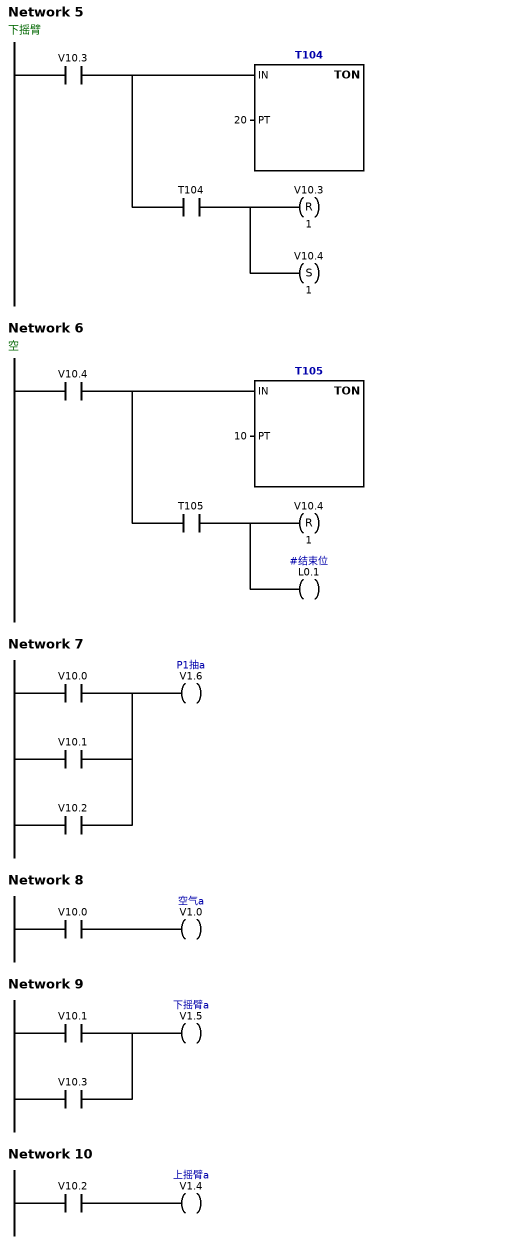
Network 5
// 下摇臂
LD     V10.3
TON    T104, 20
A      T104
R      V10.3, 1
S      V10.4, 1
Network 6
// 空
LD     V10.4
TON    T105, 10
A      T105
R      V10.4, 1
=      #结束位:L0.1
Network 7
LD     V10.0
O      V10.1
O      V10.2
=      P1抽a:V1.6
Network 8
LD     V10.0
=      空气a:V1.0
Network 9
LD     V10.1
O      V10.3
=      下摇臂a:V1.5
Network 10
LD     V10.2
=      上摇臂a:V1.4
END_SUBROUTINE_BLOCK

SUBROUTINE_BLOCK M排空:SBR5
TITLE=P1抽取比色皿内液体
VAR_INPUT
时间:WORD;	// LW0 
END_VAR
VAR_IN_OUT
启动位:BOOL;	// L2.0 
END_VAR
VAR_OUTPUT
结束位:BOOL;	// L2.1 
END_VAR
BEGIN
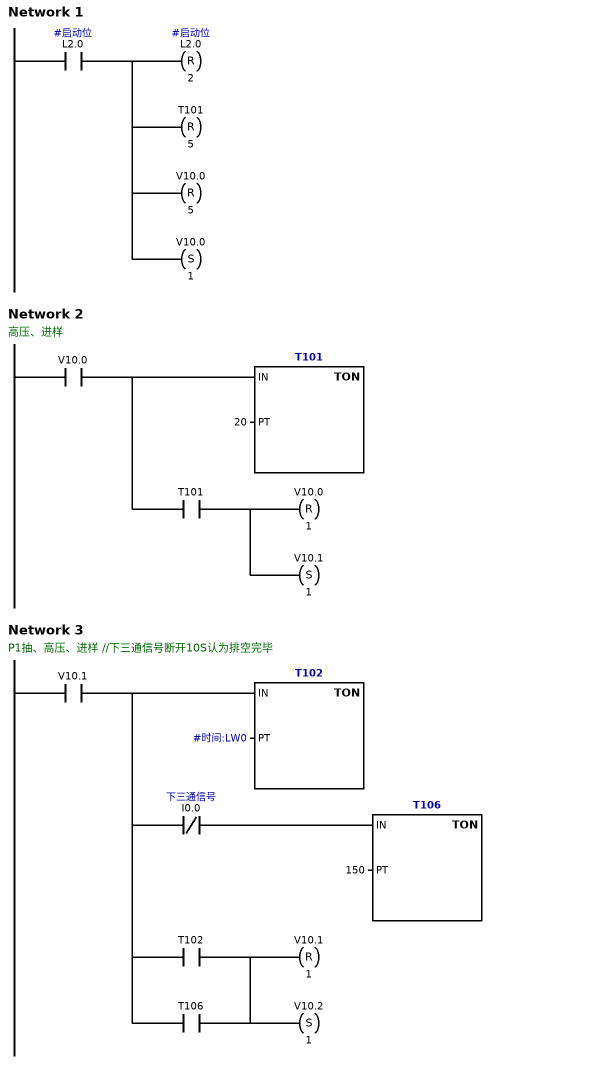
Network 1
LD     #启动位:L2.0
R      #启动位:L2.0, 2
R      T101, 5
R      V10.0, 5
S      V10.0, 1
Network 2
// 高压、进样
LD     V10.0
TON    T101, 20
A      T101
R      V10.0, 1
S      V10.1, 1
Network 3
// P1抽、高压、进样 //下三通信号断开10S认为排空完毕
LD     V10.1
LPS
TON    T102, #时间:LW0
AN     下三通信号:I0.0
TON    T106, 150
LPP
LD     T102
O      T106
ALD
R      V10.1, 1
S      V10.2, 1
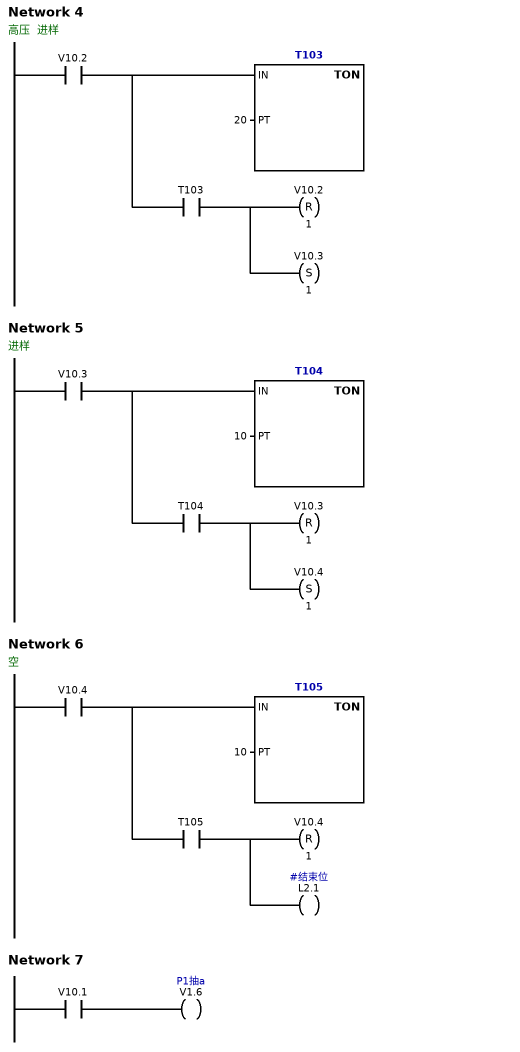
Network 4
// 高压  进样  
LD     V10.2
TON    T103, 20
A      T103
R      V10.2, 1
S      V10.3, 1
Network 5
// 进样  
LD     V10.3
TON    T104, 10
A      T104
R      V10.3, 1
S      V10.4, 1
Network 6
// 空
LD     V10.4
TON    T105, 10
A      T105
R      V10.4, 1
=      #结束位:L2.1
Network 7
LD     V10.1
=      P1抽a:V1.6
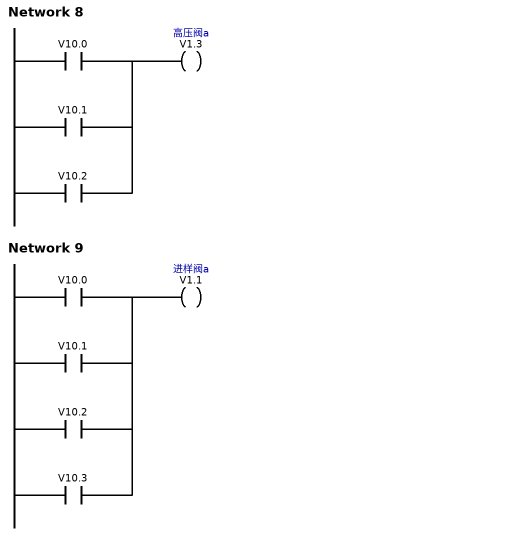
Network 8
LD     V10.0
O      V10.1
O      V10.2
=      高压阀a:V1.3
Network 9
LD     V10.0
O      V10.1
O      V10.2
O      V10.3
=      进样阀a:V1.1
END_SUBROUTINE_BLOCK

SUBROUTINE_BLOCK M润洗:SBR6
TITLE=
VAR_INPUT
抽液时间:WORD;	// LW0 
抽空时间:WORD;	// LW2 
END_VAR
VAR_IN_OUT
启动位:BOOL;	// L4.0 
END_VAR
VAR_OUTPUT
结束位:BOOL;	// L4.1 
采样阀:BOOL;	// L4.2 
END_VAR
BEGIN
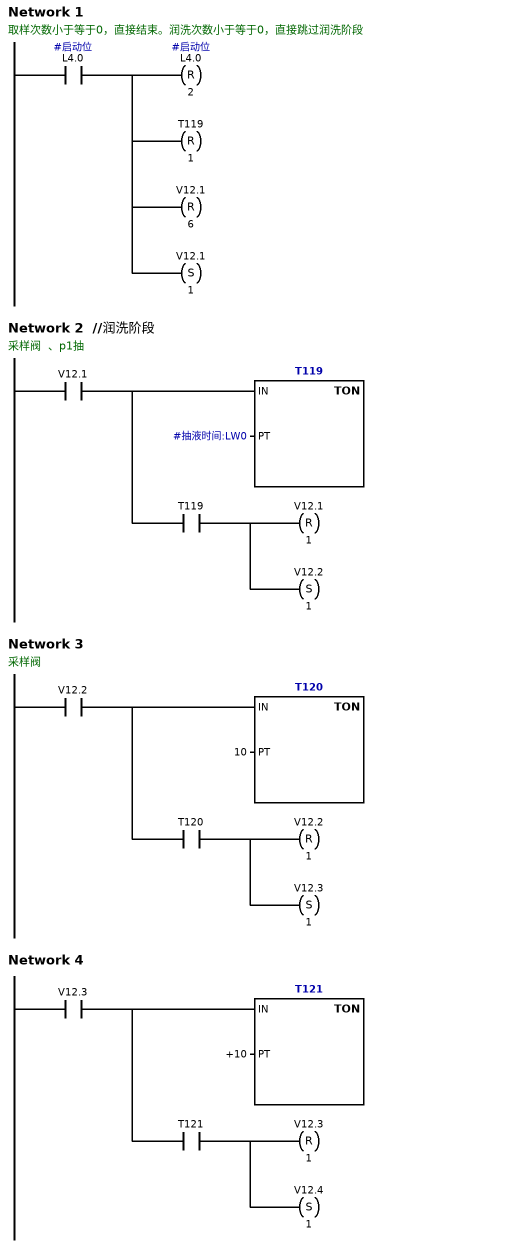
Network 1
// 取样次数小于等于0，直接结束。润洗次数小于等于0，直接跳过润洗阶段
LD     #启动位:L4.0
R      #启动位:L4.0, 2
R      T119, 1
R      V12.1, 6
S      V12.1, 1
Network 2 // //润洗阶段
// 采样阀  、p1抽
LD     V12.1
TON    T119, #抽液时间:LW0
A      T119
R      V12.1, 1
S      V12.2, 1
Network 3
//  采样阀
LD     V12.2
TON    T120, 10
A      T120
R      V12.2, 1
S      V12.3, 1
Network 4
LD     V12.3
TON    T121, +10
A      T121
R      V12.3, 1
S      V12.4, 1
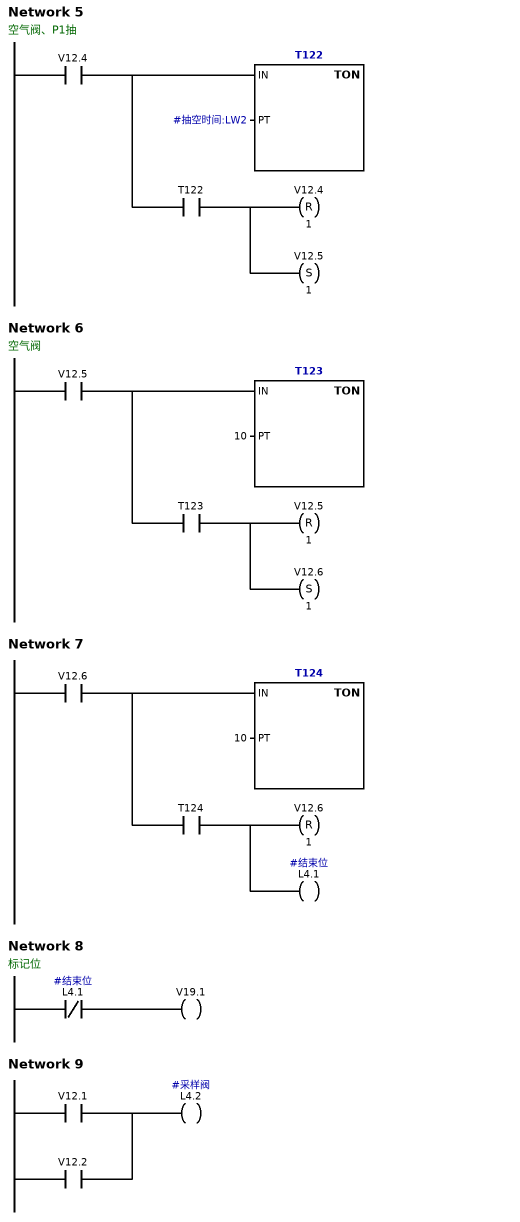
Network 5
// 空气阀、P1抽
LD     V12.4
TON    T122, #抽空时间:LW2
A      T122
R      V12.4, 1
S      V12.5, 1
Network 6
// 空气阀
LD     V12.5
TON    T123, 10
A      T123
R      V12.5, 1
S      V12.6, 1
Network 7
LD     V12.6
TON    T124, 10
A      T124
R      V12.6, 1
=      #结束位:L4.1
Network 8
// 标记位
LDN    #结束位:L4.1
=      V19.1
Network 9
LD     V12.1
O      V12.2
=      #采样阀:L4.2
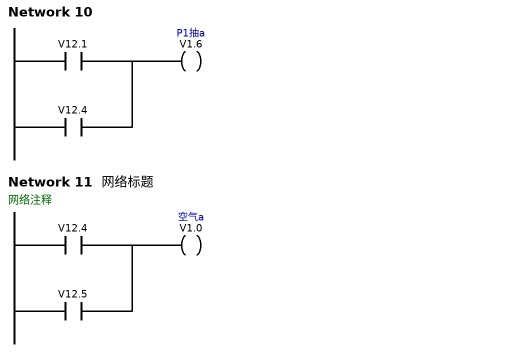
Network 10
LD     V12.1
O      V12.4
=      P1抽a:V1.6
Network 11 // 网络标题
// 网络注释
LD     V12.4
O      V12.5
=      空气a:V1.0
Network 13 // 网络标题
// 网络注释
END_SUBROUTINE_BLOCK

SUBROUTINE_BLOCK 【流程】:SBR7
TITLE=
VAR_IN_OUT
启动位:BOOL;	// L0.0 
END_VAR
VAR_OUTPUT
结束位:BOOL;	// L0.1 
END_VAR
BEGIN
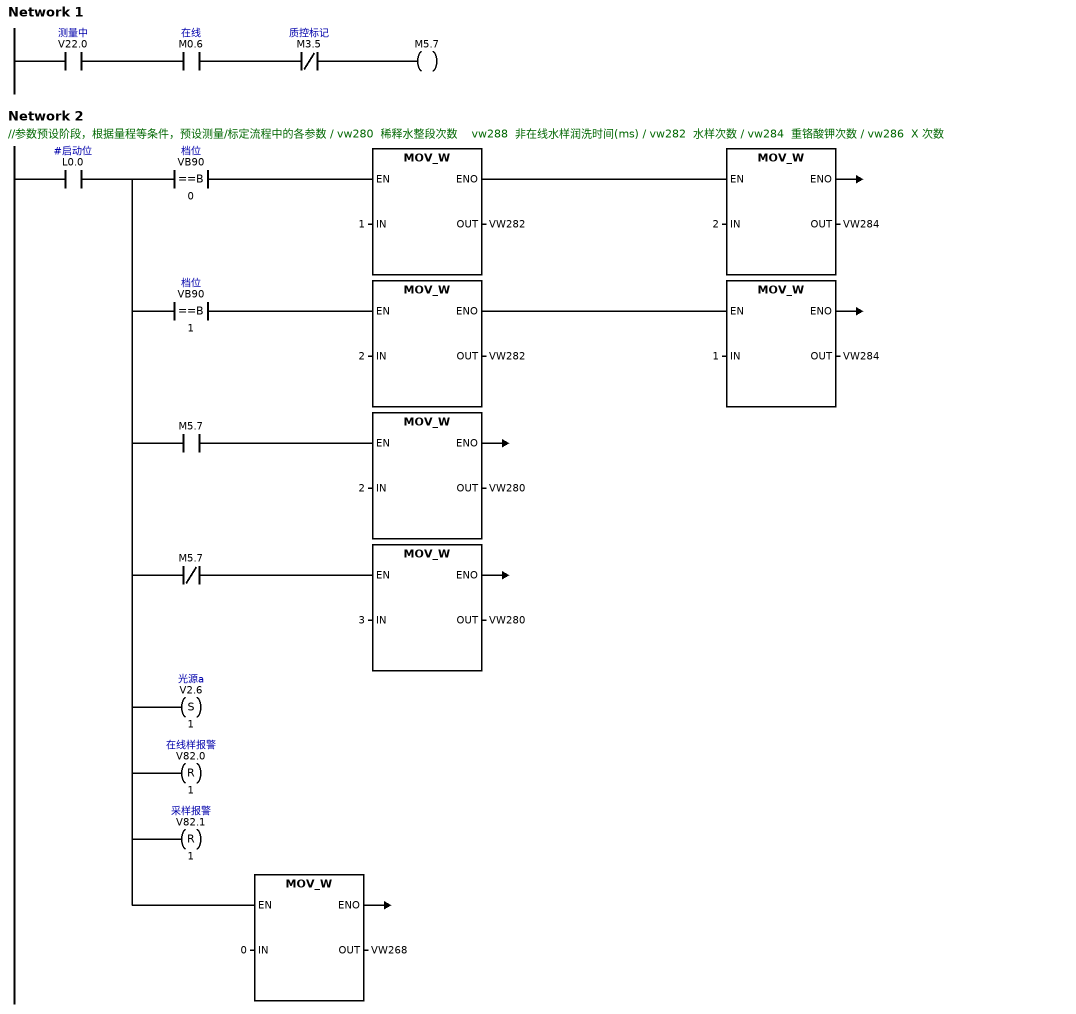
Network 1
LD     测量中:V22.0
A      在线:M0.6
AN     质控标记:M3.5
=      M5.7
Network 2
// //参数预设阶段，根据量程等条件，预设测量/标定流程中的各参数
// vw280  稀释水整段次数    vw288  非在线水样润洗时间(ms)
// vw282  水样次数
// vw284  重铬酸钾次数
// vw286  X 次数
LD     #启动位:L0.0
LPS
AB=    档位:VB90, 0
MOVW   1, VW282
AENO
MOVW   2, VW284
LRD
AB=    档位:VB90, 1
MOVW   2, VW282
AENO
MOVW   1, VW284
LRD
A      M5.7
MOVW   2, VW280
LRD
AN     M5.7
MOVW   3, VW280
LRD
S      光源a:V2.6, 1
LRD
R      在线样报警:V82.0, 1
LRD
R      采样报警:V82.1, 1
LPP
MOVW   0, VW268
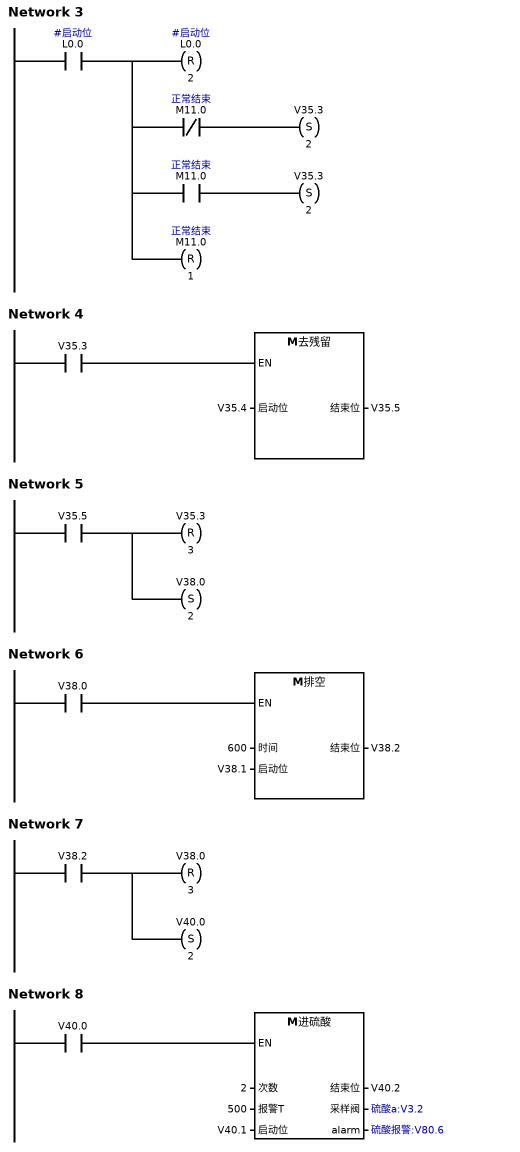
Network 3
LD     #启动位:L0.0
LPS
R      #启动位:L0.0, 2
AN     正常结束:M11.0
S      V35.3, 2
LRD
A      正常结束:M11.0
S      V35.3, 2
LPP
R      正常结束:M11.0, 1
Network 4
LD     V35.3
CALL   M去残留:SBR4, V35.4, V35.5
Network 5
LD     V35.5
R      V35.3, 3
S      V38.0, 2
Network 6
LD     V38.0
CALL   M排空:SBR5, 600, V38.1, V38.2
Network 7
LD     V38.2
R      V38.0, 3
S      V40.0, 2
Network 8
LD     V40.0
CALL   M进硫酸:SBR3, 2, 500, V40.1, V40.2, 硫酸a:V3.2, 硫酸报警:V80.6
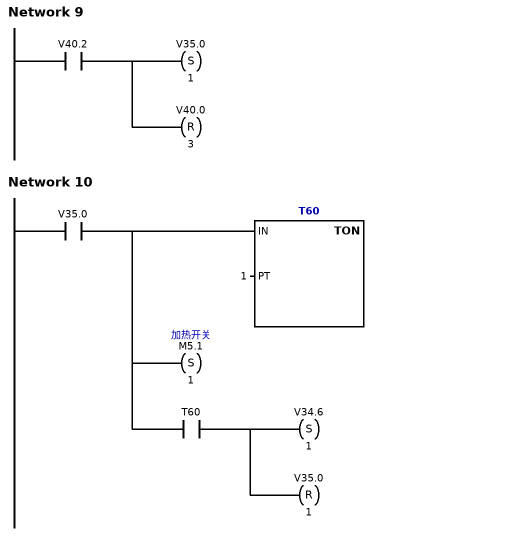
Network 9
LD     V40.2
S      V35.0, 1
R      V40.0, 3
Network 10
LD     V35.0
TON    T60, 1
S      加热开关:M5.1, 1
A      T60
S      V34.6, 1
R      V35.0, 1
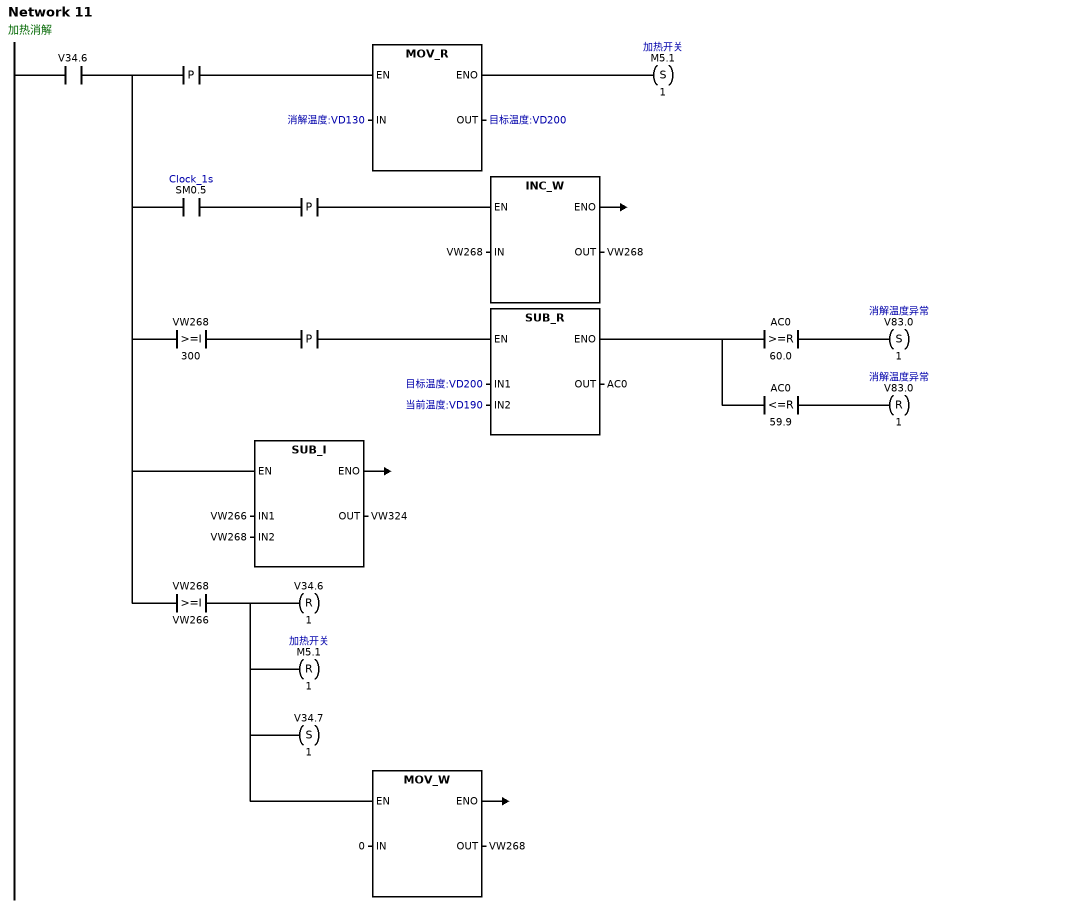
Network 11
// 加热消解
LD     V34.6
LPS
EU
MOVR   消解温度:VD130, 目标温度:VD200
AENO
S      加热开关:M5.1, 1
LRD
A      Clock_1s:SM0.5
EU
INCW   VW268
LRD
AW>=   VW268, 300
EU
MOVR   目标温度:VD200, AC0
AENO
-R     当前温度:VD190, AC0
AENO
LPS
AR>=   AC0, 60.0
S      消解温度异常:V83.0, 1
LPP
AR<=   AC0, 59.9
R      消解温度异常:V83.0, 1
LRD
MOVW   VW266, VW324
-I     VW268, VW324
LPP
AW>=   VW268, VW266
R      V34.6, 1
R      加热开关:M5.1, 1
S      V34.7, 1
MOVW   0, VW268
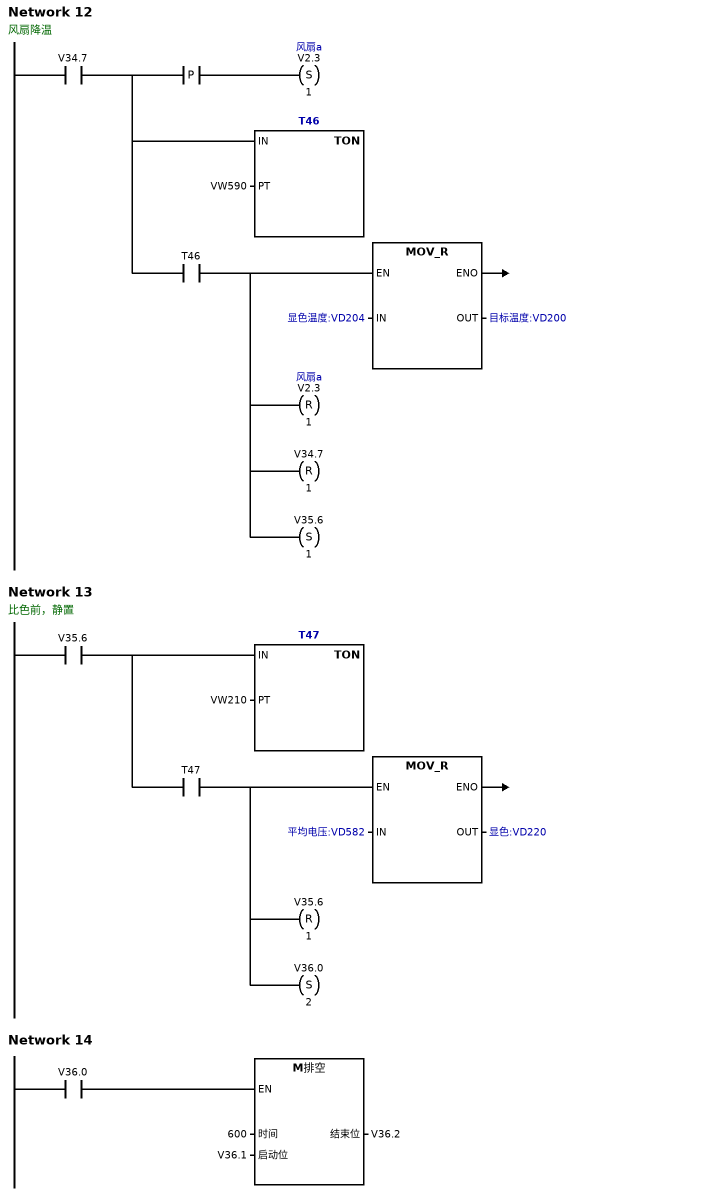
Network 12
// 风扇降温   
// (network saved uncompiled; LAD cells follow)
// row 0: c0 -| |- V34.7 v  c1 -|P|-  c2 -(S) 风扇a:V2.3, 1
// row 1: c0 ^v  c1 --  c2 [TON T46 IN:=power@row1, PT:=VW590]
// row 2: c0 ^v  c2 [box]
// row 3: c0 ^  c1 -| |- T46 v  c2 --  c3 [MOV_R EN:=power@row3, IN:=显色温度:VD204, ENO=>power, OUT=>目标温度:VD200]  c4 ->
// row 4: c1 ^v  c3 [box]
// row 5: c1 ^v  c2 -(R) 风扇a:V2.3, 1
// row 6: c1 ^v  c2 -(R) V34.7, 1
// row 7: c1 ^  c2 -(S) V35.6, 1
Network 13
// 比色前，静置
LD     V35.6
TON    T47, VW210
A      T47
MOVR   平均电压:VD582, 显色:VD220
R      V35.6, 1
S      V36.0, 2
Network 14
LD     V36.0
CALL   M排空:SBR5, 600, V36.1, V36.2
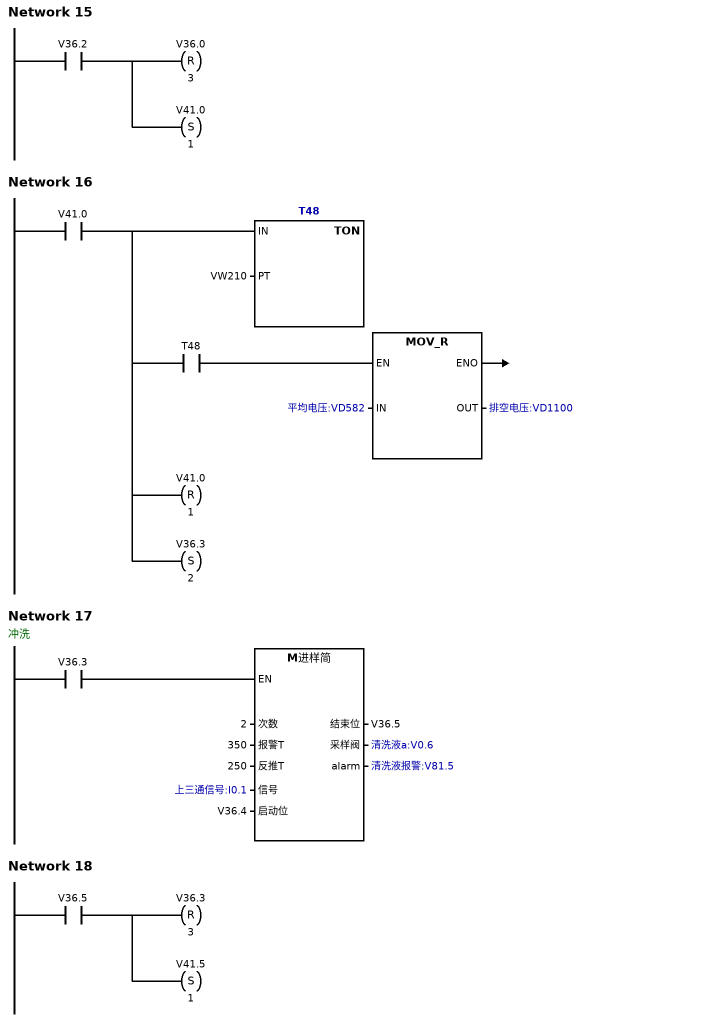
Network 15
LD     V36.2
R      V36.0, 3
S      V41.0, 1
Network 16
LD     V41.0
LPS
TON    T48, VW210
A      T48
MOVR   平均电压:VD582, 排空电压:VD1100
LRD
R      V41.0, 1
LPP
S      V36.3, 2
Network 17
// 冲洗
LD     V36.3
CALL   M进样简:SBR1, 2, 350, 250, 上三通信号:I0.1, V36.4, V36.5, 清洗液a:V0.6, 清洗液报警:V81.5
Network 18
LD     V36.5
R      V36.3, 3
S      V41.5, 1
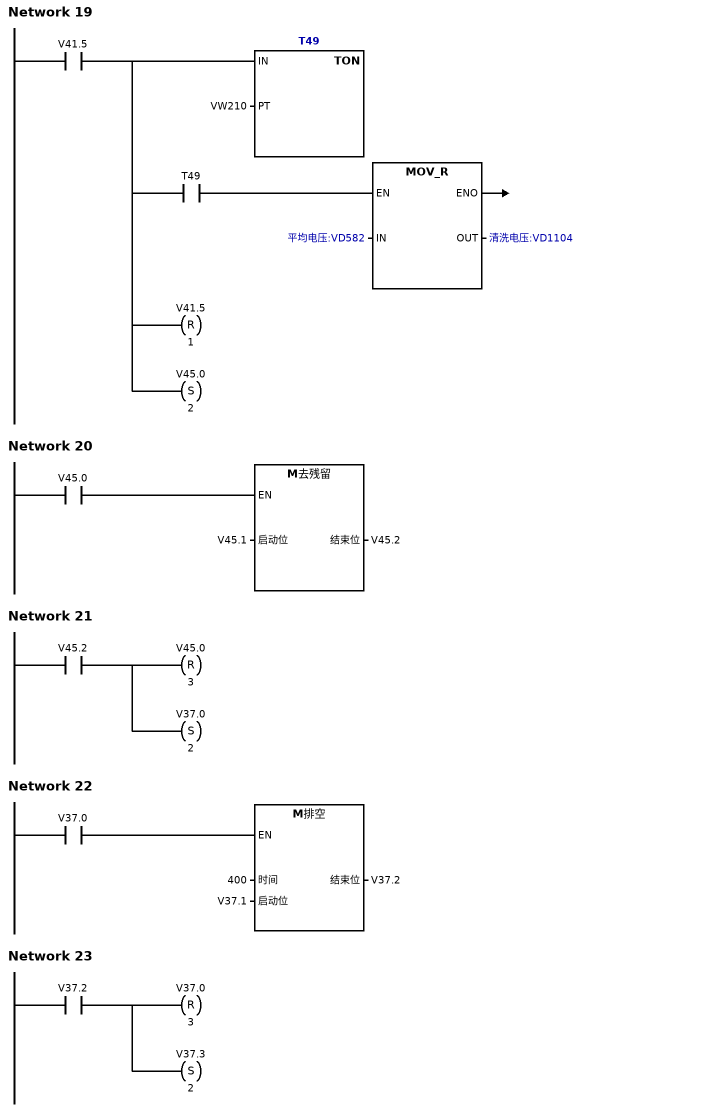
Network 19
LD     V41.5
LPS
TON    T49, VW210
A      T49
MOVR   平均电压:VD582, 清洗电压:VD1104
LRD
R      V41.5, 1
LPP
S      V45.0, 2
Network 20
LD     V45.0
CALL   M去残留:SBR4, V45.1, V45.2
Network 21
LD     V45.2
R      V45.0, 3
S      V37.0, 2
Network 22
LD     V37.0
CALL   M排空:SBR5, 400, V37.1, V37.2
Network 23
LD     V37.2
R      V37.0, 3
S      V37.3, 2
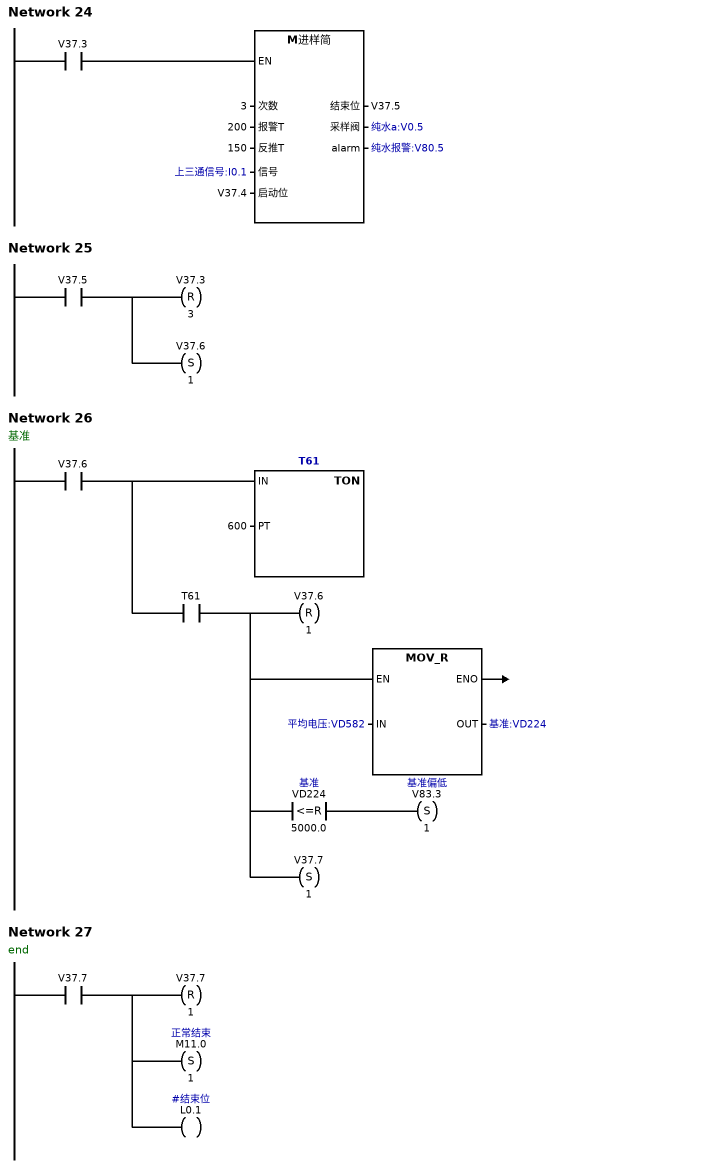
Network 24
LD     V37.3
CALL   M进样简:SBR1, 3, 200, 150, 上三通信号:I0.1, V37.4, V37.5, 纯水a:V0.5, 纯水报警:V80.5
Network 25
LD     V37.5
R      V37.3, 3
S      V37.6, 1
Network 26
// 基准
LD     V37.6
TON    T61, 600
A      T61
LPS
R      V37.6, 1
MOVR   平均电压:VD582, 基准:VD224
AR<=   基准:VD224, 5000.0
S      基准偏低:V83.3, 1
LPP
S      V37.7, 1
Network 27
// end
LD     V37.7
R      V37.7, 1
S      正常结束:M11.0, 1
=      #结束位:L0.1
END_SUBROUTINE_BLOCK

SUBROUTINE_BLOCK 输出Q:SBR8
TITLE=
BEGIN
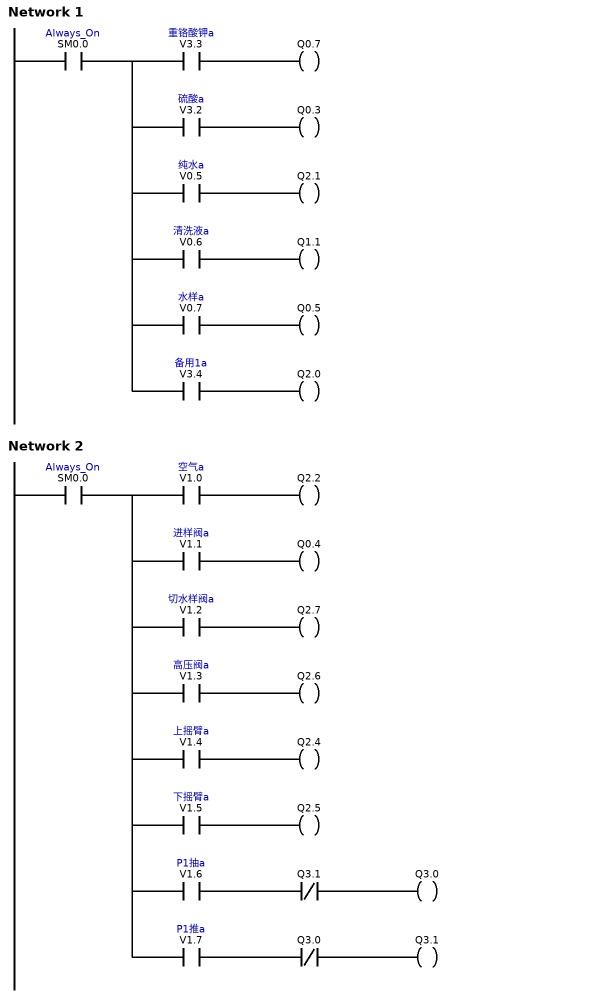
Network 1
LD     Always_On:SM0.0
LPS
A      重铬酸钾a:V3.3
=      Q0.7
LRD
A      硫酸a:V3.2
=      Q0.3
LRD
A      纯水a:V0.5
=      Q2.1
LRD
A      清洗液a:V0.6
=      Q1.1
LRD
A      水样a:V0.7
=      Q0.5
LPP
A      备用1a:V3.4
=      Q2.0
Network 2
LD     Always_On:SM0.0
LPS
A      空气a:V1.0
=      Q2.2
LRD
A      进样阀a:V1.1
=      Q0.4
LRD
A      切水样阀a:V1.2
=      Q2.7
LRD
A      高压阀a:V1.3
=      Q2.6
LRD
A      上摇臂a:V1.4
=      Q2.4
LRD
A      下摇臂a:V1.5
=      Q2.5
LRD
A      P1抽a:V1.6
AN     Q3.1
=      Q3.0
LPP
A      P1推a:V1.7
AN     Q3.0
=      Q3.1
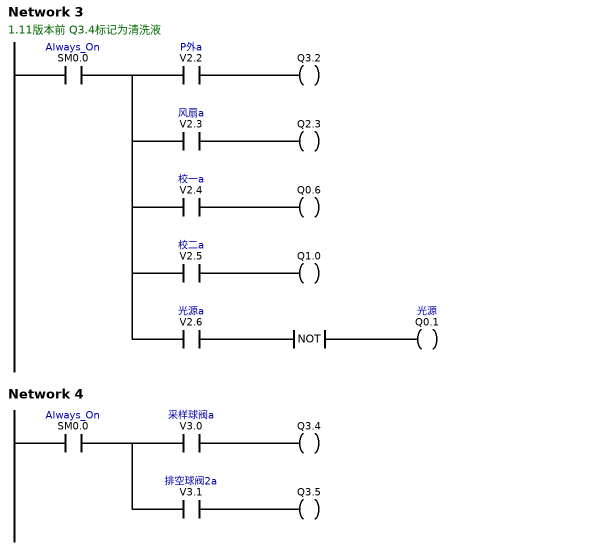
Network 3
// 1.11版本前 Q3.4标记为清洗液  
LD     Always_On:SM0.0
LPS
A      P外a:V2.2
=      Q3.2
LRD
A      风扇a:V2.3
=      Q2.3
LRD
A      校一a:V2.4
=      Q0.6
LRD
A      校二a:V2.5
=      Q1.0
LPP
A      光源a:V2.6
NOT
=      光源:Q0.1
Network 4
LD     Always_On:SM0.0
LPS
A      采样球阀a:V3.0
=      Q3.4
LPP
A      排空球阀2a:V3.1
=      Q3.5
END_SUBROUTINE_BLOCK

SUBROUTINE_BLOCK PID计算:SBR9
TITLE=子程序注释
VAR_INPUT
当前温度:REAL;	// LD0 
目标温度:REAL;	// LD4 
END_VAR
VAR_OUTPUT
占空比:INT;	// LW8 
END_VAR
VAR
温度差:REAL;	// LD10 
END_VAR
BEGIN
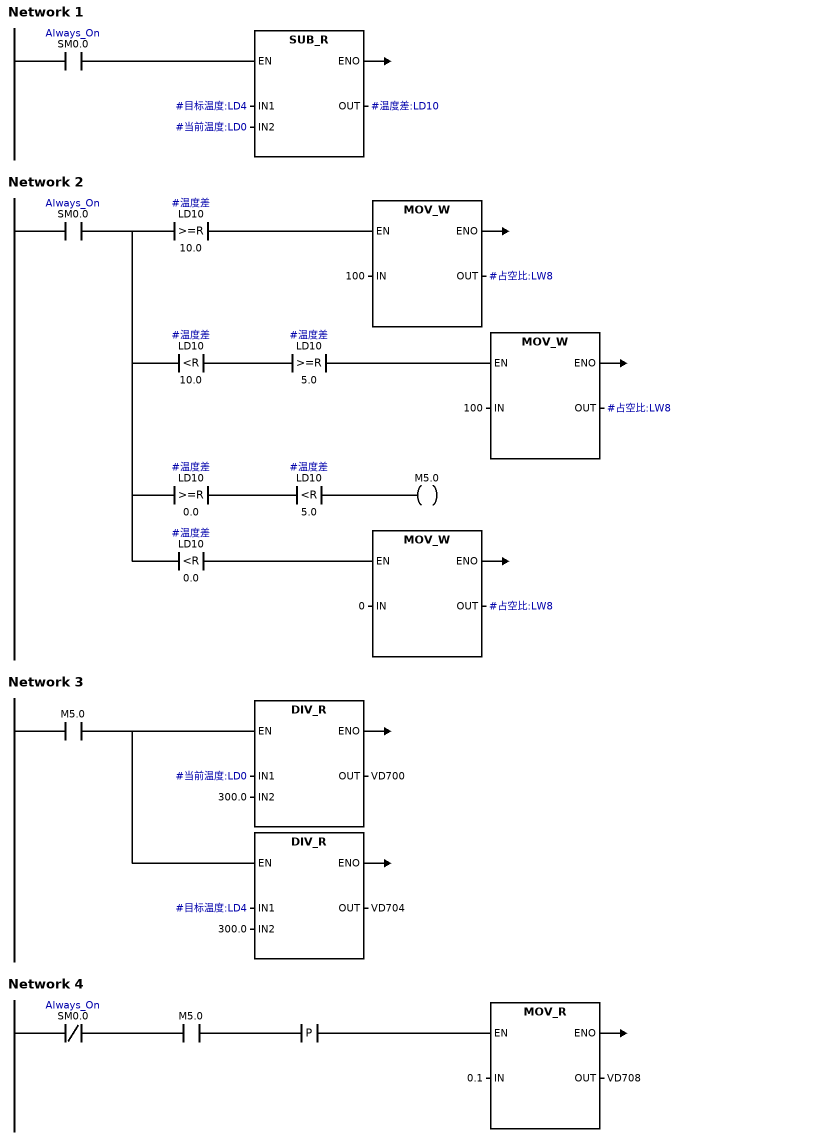
Network 1
LD     Always_On:SM0.0
MOVR   #目标温度:LD4, #温度差:LD10
-R     #当前温度:LD0, #温度差:LD10
Network 2
LD     Always_On:SM0.0
LPS
AR>=   #温度差:LD10, 10.0
MOVW   100, #占空比:LW8
LRD
AR<    #温度差:LD10, 10.0
AR>=   #温度差:LD10, 5.0
MOVW   100, #占空比:LW8
LRD
AR>=   #温度差:LD10, 0.0
AR<    #温度差:LD10, 5.0
=      M5.0
LPP
AR<    #温度差:LD10, 0.0
MOVW   0, #占空比:LW8
Network 3
LD     M5.0
MOVR   #当前温度:LD0, VD700
/R     300.0, VD700
MOVR   #目标温度:LD4, VD704
/R     300.0, VD704
Network 4
LDN    Always_On:SM0.0
A      M5.0
EU
MOVR   0.1, VD708
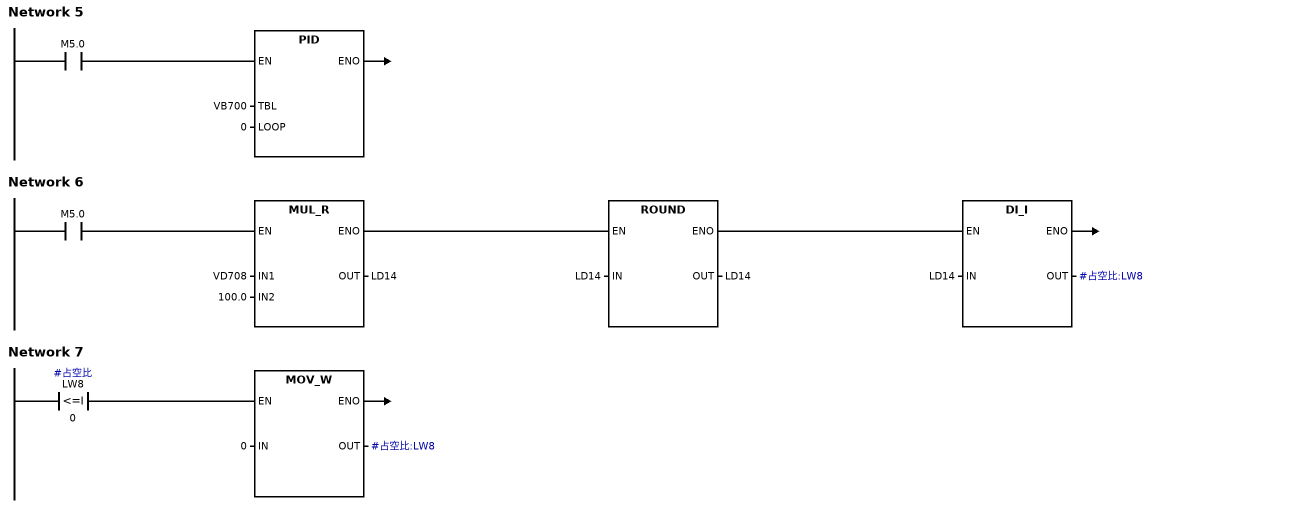
Network 5
LD     M5.0
PID    VB700, 0
Network 6
LD     M5.0
MOVR   VD708, LD14
AENO
*R     100.0, LD14
AENO
ROUND  LD14, LD14
AENO
DTI    LD14, #占空比:LW8
Network 7
LDW<=  #占空比:LW8, 0
MOVW   0, #占空比:LW8
END_SUBROUTINE_BLOCK

SUBROUTINE_BLOCK 二层:SBR10
TITLE=子程序注释
BEGIN
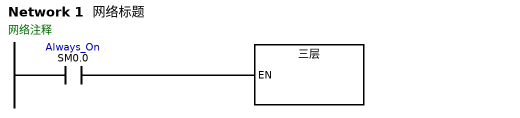
Network 1 // 网络标题
// 网络注释
LD     Always_On:SM0.0
CALL   三层:SBR36
END_SUBROUTINE_BLOCK

SUBROUTINE_BLOCK KBA:SBR11
TITLE=子程序注释
VAR_INPUT
显色1:REAL;	// LD0 
基准1:REAL;	// LD4 
浓度1:REAL;	// LD8 
显色2:REAL;	// LD12 
基准2:REAL;	// LD16 
浓度2:REAL;	// LD20 
END_VAR
VAR_OUTPUT
A1:REAL;	// LD24 
A2:REAL;	// LD28 
K:REAL;	// LD32 
b:REAL;	// LD36 
END_VAR
BEGIN
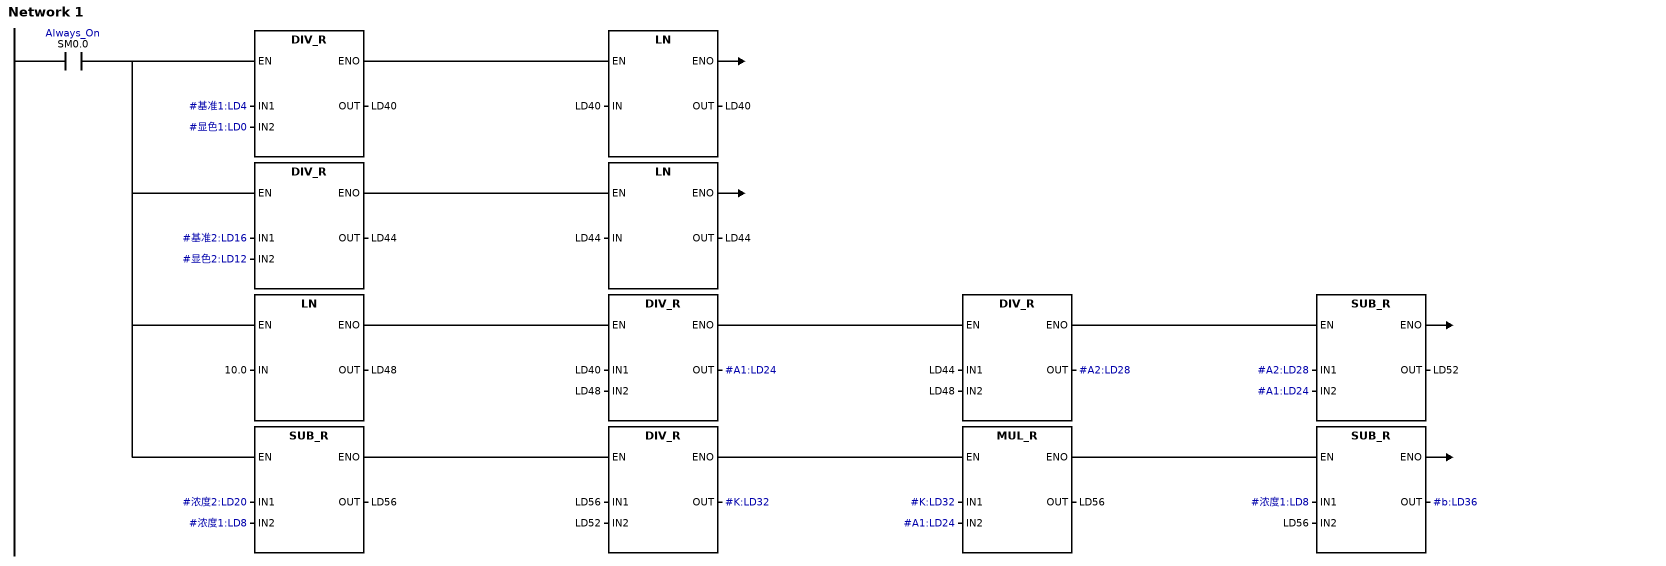
Network 1
LD     Always_On:SM0.0
LPS
MOVR   #基准1:LD4, LD40
AENO
/R     #显色1:LD0, LD40
AENO
LN     LD40, LD40
LRD
MOVR   #基准2:LD16, LD44
AENO
/R     #显色2:LD12, LD44
AENO
LN     LD44, LD44
LRD
LN     10.0, LD48
AENO
MOVR   LD40, #A1:LD24
AENO
/R     LD48, #A1:LD24
AENO
MOVR   LD44, #A2:LD28
AENO
/R     LD48, #A2:LD28
AENO
MOVR   #A2:LD28, LD52
-R     #A1:LD24, LD52
LPP
MOVR   #浓度2:LD20, LD56
AENO
-R     #浓度1:LD8, LD56
AENO
MOVR   LD56, #K:LD32
AENO
/R     LD52, #K:LD32
AENO
MOVR   #K:LD32, LD56
AENO
*R     #A1:LD24, LD56
AENO
MOVR   #浓度1:LD8, #b:LD36
-R     LD56, #b:LD36
Network 2 // 网络标题
// 网络注释
END_SUBROUTINE_BLOCK

SUBROUTINE_BLOCK 间隔测量:SBR12
TITLE=子程序注释
BEGIN
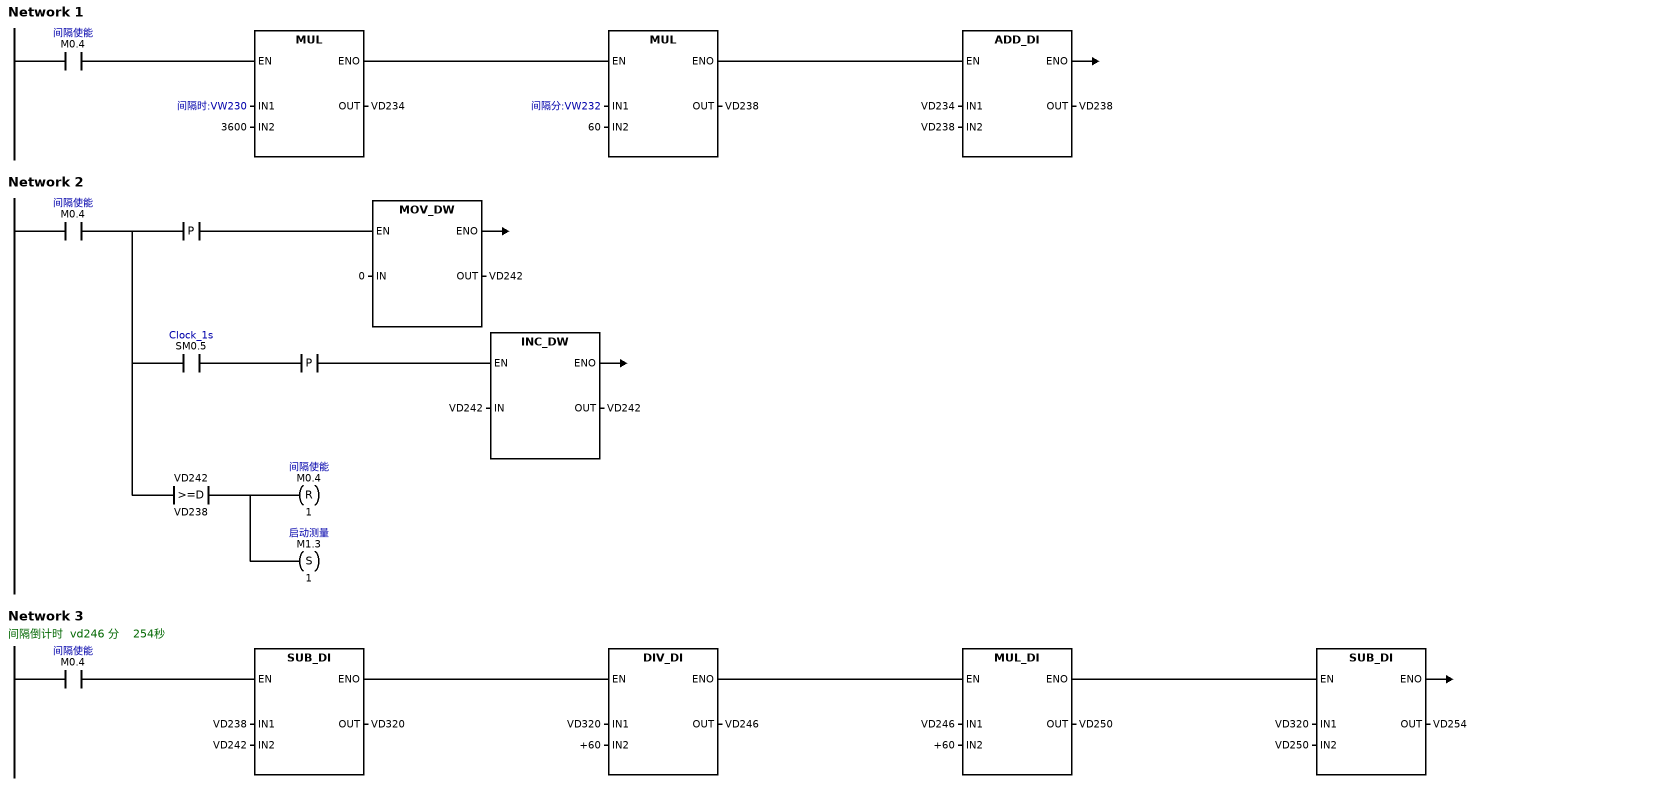
Network 1
LD     间隔使能:M0.4
MOVW   间隔时:VW230, VW236
AENO
MUL    3600, VD234
AENO
MOVW   间隔分:VW232, VW240
AENO
MUL    60, VD238
AENO
+D     VD234, VD238
Network 2
LD     间隔使能:M0.4
LPS
EU
MOVD   0, VD242
LRD
A      Clock_1s:SM0.5
EU
INCD   VD242
LPP
AD>=   VD242, VD238
R      间隔使能:M0.4, 1
S      启动测量:M1.3, 1
Network 3
// 间隔倒计时  vd246 分    254秒
LD     间隔使能:M0.4
MOVD   VD238, VD320
AENO
-D     VD242, VD320
AENO
MOVD   VD320, VD246
AENO
/D     +60, VD246
AENO
MOVD   VD246, VD250
AENO
*D     +60, VD250
AENO
MOVD   VD320, VD254
-D     VD250, VD254
Network 4 // 网络标题
// 网络注释
END_SUBROUTINE_BLOCK

SUBROUTINE_BLOCK 整点测量:SBR13
TITLE=子程序注释
BEGIN
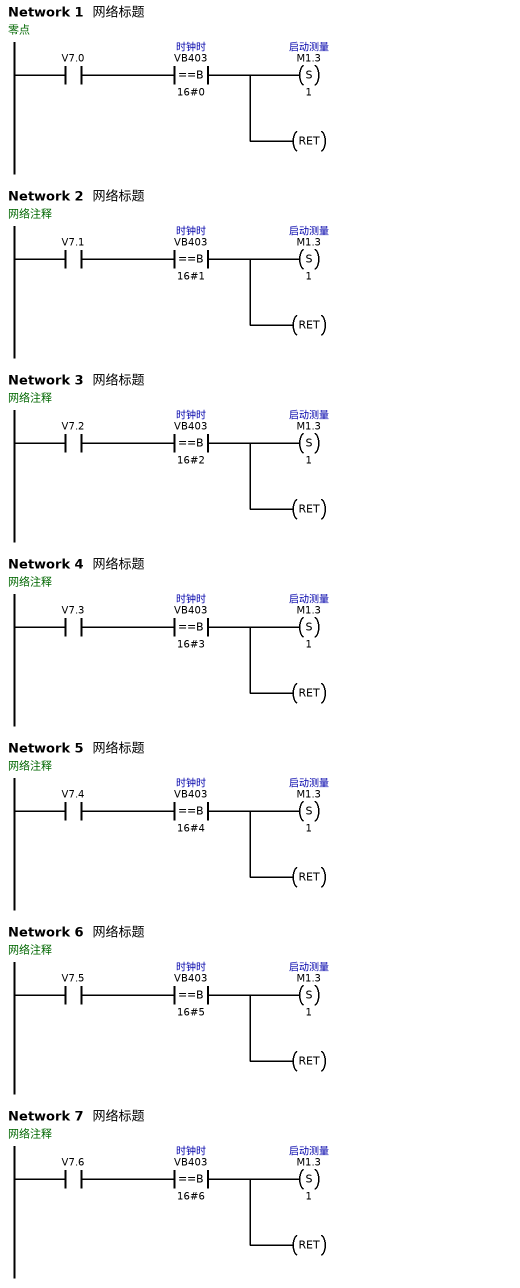
Network 1 // 网络标题
// 零点
LD     V7.0
AB=    时钟时:VB403, 16#0
S      启动测量:M1.3, 1
CRET
Network 2 // 网络标题
// 网络注释
LD     V7.1
AB=    时钟时:VB403, 16#1
S      启动测量:M1.3, 1
CRET
Network 3 // 网络标题
// 网络注释
LD     V7.2
AB=    时钟时:VB403, 16#2
S      启动测量:M1.3, 1
CRET
Network 4 // 网络标题
// 网络注释
LD     V7.3
AB=    时钟时:VB403, 16#3
S      启动测量:M1.3, 1
CRET
Network 5 // 网络标题
// 网络注释
LD     V7.4
AB=    时钟时:VB403, 16#4
S      启动测量:M1.3, 1
CRET
Network 6 // 网络标题
// 网络注释
LD     V7.5
AB=    时钟时:VB403, 16#5
S      启动测量:M1.3, 1
CRET
Network 7 // 网络标题
// 网络注释
LD     V7.6
AB=    时钟时:VB403, 16#6
S      启动测量:M1.3, 1
CRET
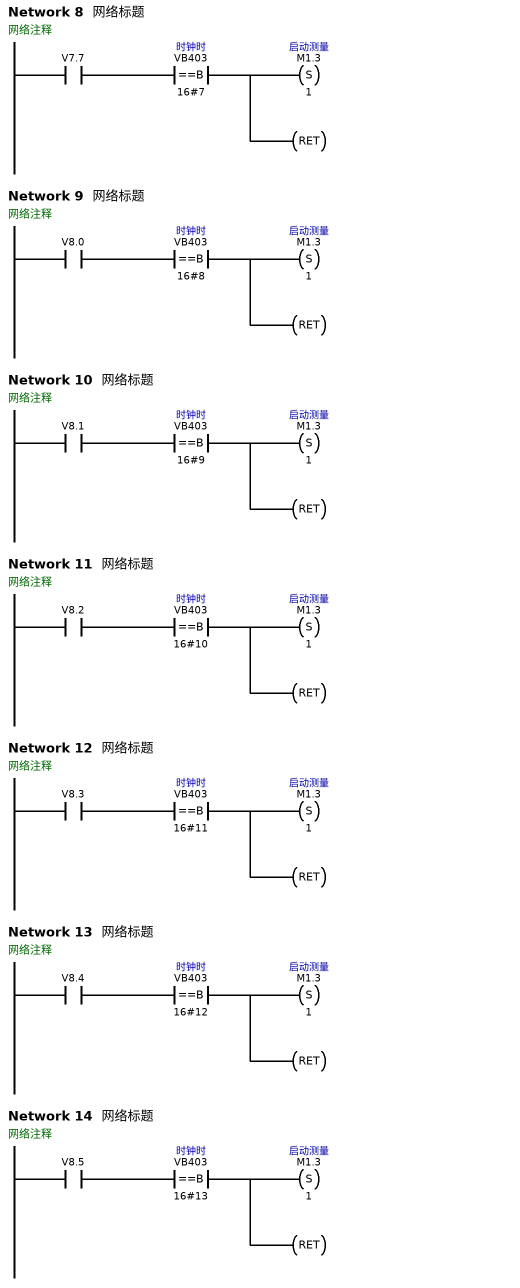
Network 8 // 网络标题
// 网络注释
LD     V7.7
AB=    时钟时:VB403, 16#7
S      启动测量:M1.3, 1
CRET
Network 9 // 网络标题
// 网络注释
LD     V8.0
AB=    时钟时:VB403, 16#8
S      启动测量:M1.3, 1
CRET
Network 10 // 网络标题
// 网络注释
LD     V8.1
AB=    时钟时:VB403, 16#9
S      启动测量:M1.3, 1
CRET
Network 11 // 网络标题
// 网络注释
LD     V8.2
AB=    时钟时:VB403, 16#10
S      启动测量:M1.3, 1
CRET
Network 12 // 网络标题
// 网络注释
LD     V8.3
AB=    时钟时:VB403, 16#11
S      启动测量:M1.3, 1
CRET
Network 13 // 网络标题
// 网络注释
LD     V8.4
AB=    时钟时:VB403, 16#12
S      启动测量:M1.3, 1
CRET
Network 14 // 网络标题
// 网络注释
LD     V8.5
AB=    时钟时:VB403, 16#13
S      启动测量:M1.3, 1
CRET
